# B&R Automation Studio project Sim_Eksamen_Test
Automation Studio 4.7.2.98

## Configuration X20CP1382

### Hardware
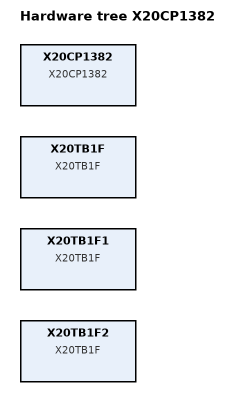
```
X20CP1382 : X20CP1382 v1.8.0.0  [X1 -> X1.SL; X2 -> X2.SL; X3 -> X3.SL]
  Module X1 (Type=X1, Virtual=true, Version=1.8.0.0)
    Connection (Connector=SS1, TargetModule=X20TB1F, TargetConnector=SS)
    Connection (Connector=SL, TargetModule=X20CP1382, TargetConnector=X1)
  Module X2 (Type=X2, Virtual=true, Version=1.8.0.0)
    Connection (Connector=SS1, TargetModule=X20TB1F1, TargetConnector=SS)
    Connection (Connector=SL, TargetModule=X20CP1382, TargetConnector=X2)
  Module X3 (Type=X3, Virtual=true, Version=1.8.0.0)
    Connection (Connector=SS1, TargetModule=X20TB1F2, TargetConnector=SS)
    Connection (Connector=SL, TargetModule=X20CP1382, TargetConnector=X3)
  Connector IF2:
    ActivateDevice = 1
  ConfigurationID = Sim_Eksamen_Test_X20CP1382
  Simulation = 1
X20TB1F : X20TB1F v1.0.0.0
X20TB1F1 : X20TB1F v1.0.0.0
X20TB1F2 : X20TB1F v1.0.0.0
```

## Logical view

### Global.typ
```iecst
(*Denne Type er de 3 stadier som vores robot arm kan befinde sig i.*)

TYPE
	RobotArm : 	STRUCT
		Home : BOOL;
		Getting : BOOL;
		Delivering : BOOL;
	END_STRUCT;
END_TYPE
```

### Global.var
```iecst
VAR
	diGoBtn : BOOL;
END_VAR

VAR CONSTANT

END_VAR
```

### Program Logical/Feed_Conv

#### Variables.var
```iecst
VAR
	TON_Timer : TON;
	doConvSideStart : BOOL;
	doFeederMid : BOOL;
	doFeederLeft : BOOL;
	doFeederRight : BOOL;
	doConvMainStart : BOOL;
	FeedCount : USINT;
END_VAR
```

#### Main.st
```iecst
PROGRAM _INIT
	// Feeder timer initialization
	TON_Timer.PT := T#2s;

END_PROGRAM

PROGRAM _CYCLIC

	IF diGoBtn THEN
		doConvMainStart := TRUE;
		TON_Timer.IN := TRUE;

		// Johans Feeder roundtable.
		IF FeedCount = 0 AND TON_Timer.Q THEN
			doFeederLeft := TRUE;
			doFeederRight := FALSE;
			FeedCount := 1;
			TON_Timer.IN := FALSE;
		ELSIF FeedCount = 1 AND TON_Timer.Q THEN
			doFeederMid := TRUE;
			doFeederLeft := FALSE;
			FeedCount := 2;
			TON_Timer.IN := FALSE;
		ELSIF FeedCount = 2 AND TON_Timer.Q THEN
			doFeederRight := TRUE;
			doFeederMid := FALSE;
			TON_Timer.IN := FALSE;
			FeedCount := 0;
		END_IF;

	ELSE
		// Reset all.
		doConvMainStart := FALSE;
		doFeederLeft := FALSE;
		doFeederMid := FALSE;
		doFeederRight := FALSE;
		TON_Timer.IN := FALSE;
	END_IF;

	// Functionblock Calls
	TON_Timer();
END_PROGRAM

PROGRAM _EXIT
	(* Insert code here *)

END_PROGRAM
```

### Program Logical/Stacker

#### Variables.var
```iecst
VAR
	diPickingSensor : BOOL;
	doStackerRight : BOOL;
	doStackerLeft : BOOL;
	doStackerPick : BOOL;
	Stacked : BOOL;
	R_TRIG_diGoBtn : R_TRIG;
	pickerRobotRight : RobotArm;
	pickerRobotLeft : RobotArm;
	R_TRIG_StackerCount : R_TRIG;
	R_TRIG_Stacked : R_TRIG;
	doConvSideStart : BOOL;
	diPlateBoxBlocked : BOOL;
	F_TRIG_BoxBlocked : F_TRIG;
	doStackerInputBelt : BOOL;
	diStackerInputSensor : BOOL;
	stackCount : USINT;
END_VAR
```

#### Main.st
```iecst
PROGRAM _INIT
	// Timer initialization
END_PROGRAM

PROGRAM _CYCLIC
	R_TRIG_Stacked.CLK := Stacked;
	R_TRIG_diGoBtn.CLK := diGoBtn;
	F_TRIG_BoxBlocked.CLK := diPlateBoxBlocked;
	R_TRIG_StackerCount.CLK := diStackerInputSensor;

	IF diGoBtn THEN
		// Stop belt when box is exactly in place.
		doStackerInputBelt := NOT diStackerInputSensor;

		// Activate stackers
		IF diStackerInputSensor THEN
			// Increase count on rising edge
			IF R_TRIG_StackerCount.Q THEN
	  			stackCount := stackCount +1;
			END_IF;

			doStackerPick := NOT (stackCount > 8) AND NOT doConvSideStart;
		ELSE
			doStackerPick := FALSE;
		END_IF;

		// Initiate plate serving
		IF R_TRIG_diGoBtn.Q THEN
			doConvSideStart := TRUE;
		END_IF;

		// Move output belt when the stack is stacked, and stop it again.
		IF R_TRIG_Stacked.Q THEN
			doConvSideStart := TRUE;
		END_IF;
		IF F_TRIG_BoxBlocked.Q THEN
			doConvSideStart := FALSE;
			// Reset count according to wether a block is ready for pickup or not
			IF diStackerInputSensor THEN
				stackCount := 1;
			ELSE
				stackCount := 0;
			END_IF;
		END_IF;

	ELSE
		// Reset all.
		doStackerPick := FALSE;
		doConvSideStart := FALSE;
		doStackerInputBelt := FALSE;
		stackCount := 0;
	END_IF;

	// Functionblock Calls
	R_TRIG_Stacked();
	R_TRIG_diGoBtn();
	F_TRIG_BoxBlocked();
	R_TRIG_StackerCount();
END_PROGRAM

PROGRAM _EXIT
	(* Insert code here *)

END_PROGRAM
```
